Staubli VAL3: Init.pgx

program Init()
  local num l_ni
begin
  //
  bExit=false
  bUserRefresh=true
  PublicData:sStatus="stop"
end
